(* IEC 61131-3 sources: AXOpen/src/data/app/src, 2 files *)

(* ---- configuration.st ---- *)
USING AXOpen.Data;
CONFIGURATION MyConfiguration
    TASK Main(Interval := T#10ms, Priority := 1);
    PROGRAM P1 WITH Main: MyProgram;

    VAR_GLOBAL
        {S7.extern=ReadWrite}
        _rtc : AXOpen.S71500.Rtc;
        {S7.extern=ReadWrite}
        _rtm : AXOpen.S71500.Rtm;

        {S7.extern=ReadWrite}
        AxoDataExchangeContext : AxoDataExchangeExample.Context;
        {S7.extern=ReadWrite}
        AxoDataFragmentsExchangeContext : AxoDataFramentsExchangeExample.Context;
        {S7.extern=ReadWrite}
        AxoDataPersistentContext : AxoDataPersistentExchangeExample.Context;
        {S7.extern=ReadWrite}
        AxoDataDistributedContext : AxoDataDistributedExample.Context;

    END_VAR
END_CONFIGURATION

(* ---- program.st ---- *)
PROGRAM MyProgram
    VAR_EXTERNAL
        _rtc : AXOpen.S71500.Rtc;
        _rtm : AXOpen.S71500.Rtm;
        AxoDataExchangeContext : AxoDataExchangeExample.Context;
        AxoDataFragmentsExchangeContext : AxoDataFramentsExchangeExample.Context;
        AxoDataPersistentContext : AxoDataPersistentExchangeExample.Context;
        AxoDataDistributedContext : AxoDataDistributedExample.Context;
    END_VAR

    AxoDataExchangeContext.InjectRtc(_rtc);
    AxoDataExchangeContext.InjectRtm(_rtm);
    AxoDataExchangeContext.Run();

    AxoDataFragmentsExchangeContext.InjectRtc(_rtc);
    AxoDataFragmentsExchangeContext.InjectRtm(_rtm);
    AxoDataFragmentsExchangeContext.Run();

    AxoDataPersistentContext.InjectRtc(_rtc);
    AxoDataPersistentContext.InjectRtm(_rtm);
    AxoDataPersistentContext.Run();

    AxoDataDistributedContext.InjectRtc(_rtc);
    AxoDataDistributedContext.InjectRtm(_rtm);
    AxoDataDistributedContext.Run();
END_PROGRAM
